PROGRAM MAIN
VAR
END_VAR

PrgMqttCom();

END_PROGRAM

(* stored: Version 1.1.0.1, ProductVersion 3.1.4022.3
   POU MAIN: Id {30044325-b307-40b2-a424-0be815c9fdc2}, SpecialFunc None *)
